// TIA Portal V17 export
// export: Created 2024-06-14T09:53:08.5091314Z, ExportSetting WithDefaults, DisplayName Totally Integrated Automation Portal, DisplayVersion V17, DisplayName TIA Portal Openness, DisplayVersion V17, DisplayName TIA Portal Version Control Interface, DisplayVersion V17, DisplayName Simotion SCOUT TIA, DisplayVersion 5.4.3.0, DisplayName SINAMICS Startdrive Advanced, DisplayVersion V17 SP1 Update 1, DisplayName SINAMICS Startdrive G110M, G120, G120C, G120D, G120P, G115D, DisplayVersion V17 SP1 Update 1, DisplayName SINAMICS Startdrive G130, G150, S120, S150, SINAMICS MV, S210, DisplayVersion V17 SP1 Update 1, DisplayName STEP 7 Professional, DisplayVersion V17, DisplayName STEP 7 Safety, DisplayVersion V17, DisplayName WinCC Professional, DisplayVersion V17
FUNCTION_BLOCK "Check_scale_LPG"   // FB7, LAD
{ S7_Optimized_Access := 'TRUE' }
VERSION : 0.1
// stored: AutoNumber true, IsIECCheckEnabled false, IsRetainMemResEnabled false, MemoryReserve 100, SetENOAutomatically false, UDAEnableTagReadback false
   VAR_INPUT
      Stopper_sesnor : Bool;
      Cylinder_presence : Bool;
      Pass_line_jammer : Bool;
      Down_line_jammer : Bool;
      Start_cycle : Bool;
      Reset_Cycle : Bool;
      Result : Int;
      Pusher : Bool;
      all_fill_done : Bool;
      xResult : Bool;
   END_VAR
   VAR_OUTPUT
      Stopper : Bool;
      LiftTable : Bool;
      Start_Check_Scale : Bool;
      Divider : Bool;
      Reset : Bool;
      CYCLE_ONE : Bool;
   END_VAR
   VAR
      Check_Scale_Started : Bool;
      Lift_Table { S7_SetPoint := 'True'} : TON_TIME;
      PASS : Bool;
      FAIL : Bool;
      LIFT_down { S7_SetPoint := 'True'} : TON_TIME;
      Temp_1 : Int;
      p_trig : Array[0..10] of Bool;
   END_VAR
   VAR RETAIN
      Stopper_count { S7_SetPoint := 'True'} : CTU_INT;
   END_VAR
   VAR
      counter_reset : Bool;
      Scale { S7_SetPoint := 'True'} : TON_TIME;
      Pusher_reset { S7_SetPoint := 'True'} : TON_TIME;
      datasend { ExternalAccessible := 'False'; ExternalVisible := 'False'; ExternalWritable := 'False'} : Bool;
      fb_Fifo_Instance { S7_SetPoint := 'True'} : "fb_Fifo";
      idx7 : Int;
      fb_Compress_Instance { S7_SetPoint := 'True'} : "fb_Compress";
      jammer_on { S7_SetPoint := 'True'} : TON_TIME;
      jammer : Bool;
      pusher_enable : Bool;
      Scale_done : Bool;
   END_VAR
   VAR RETAIN
      Lift_Table_UP { S7_SetPoint := 'True'} : CTU_INT;
   END_VAR
   VAR
      fb_Fifo_Instance_1 { S7_SetPoint := 'True'} : "fb_Fifo";
      fb_Compress_Instance_1 { S7_SetPoint := 'True'} : "fb_Compress";
      timer_1 { S7_SetPoint := 'True'} : TON_TIME;
   END_VAR
   VAR_TEMP
      temp : Int;
   END_VAR
   VAR_TEMP   // added for the SCL form of the ladder/FBD networks
      _w1 : Bool;
      _w2 : Bool;
   END_VAR
BEGIN

REGION Network 1
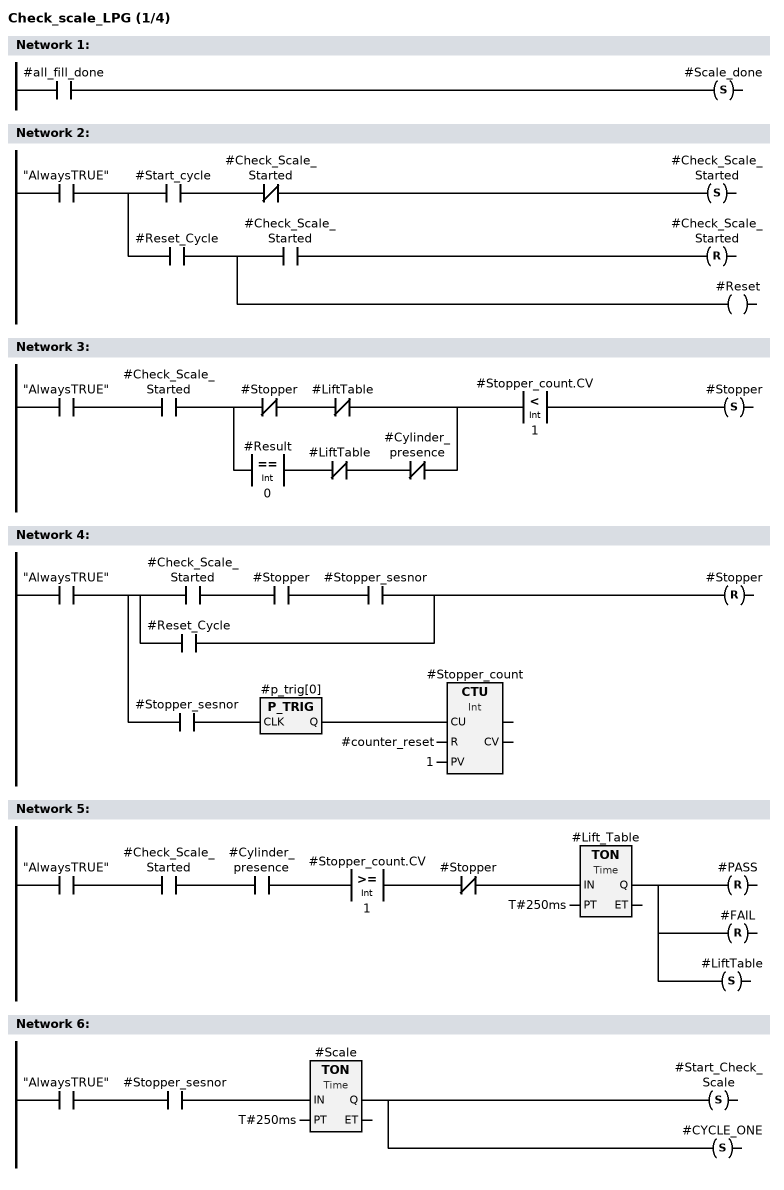
   RUNG wire#powerrail
      Contact( #all_fill_done )
      S_Coil( #Scale_done )
   END_RUNG
   // the same network as SCL:
   IF #all_fill_done THEN #Scale_done := TRUE; END_IF;
END_REGION

REGION Network 2
   RUNG wire#powerrail
      Contact( "AlwaysTRUE" )
      wire#w1
      Contact( #Start_cycle )
      I_Contact( #Check_Scale_Started )
      S_Coil( #Check_Scale_Started )
   END_RUNG
   RUNG wire#w1
      Contact( #Reset_Cycle )
      wire#w2
      Contact( #Check_Scale_Started )
      R_Coil( #Check_Scale_Started )
   END_RUNG
   RUNG wire#w2
      Coil( #Reset )
   END_RUNG
   // the same network as SCL:
   IF "AlwaysTRUE" AND #Start_cycle AND NOT #Check_Scale_Started THEN #Check_Scale_Started := TRUE; END_IF;
   #_w1 := "AlwaysTRUE" AND #Reset_Cycle;
   IF #_w1 AND #Check_Scale_Started THEN #Check_Scale_Started := FALSE; END_IF;
   #Reset := #_w1;
END_REGION

REGION Network 3
   RUNG wire#powerrail
      Contact( "AlwaysTRUE" )
      Contact( #Check_Scale_Started )
      wire#w1
      I_Contact( #Stopper )
      I_Contact( #LiftTable )
      wire#w2
      { S7_Templates := "SrcType := Int" } LT_Contact(in1 := #Stopper_count.CV, in2 := 1)
      S_Coil( #Stopper )
   END_RUNG
   RUNG wire#w1
      { S7_Templates := "SrcType := Int" } EQ_Contact(in1 := #Result, in2 := 0)
      I_Contact( #LiftTable )
      I_Contact( #Cylinder_presence )
   END_RUNG wire#w2
   // the same network as SCL:
   IF "AlwaysTRUE" AND #Check_Scale_Started AND ((NOT #Stopper AND NOT #LiftTable) OR ((#Result = 0) AND NOT #LiftTable AND NOT #Cylinder_presence)) AND (#Stopper_count.CV < 1) THEN
       #Stopper := TRUE;
   END_IF;
END_REGION

REGION Network 4
   RUNG wire#powerrail
      Contact( "AlwaysTRUE" )
      wire#w1
      Contact( #Check_Scale_Started )
      Contact( #Stopper )
      Contact( #Stopper_sesnor )
      wire#w2
      R_Coil( #Stopper )
   END_RUNG
   RUNG wire#w1
      Contact( #Reset_Cycle )
   END_RUNG wire#w2
   RUNG wire#w1
      Contact( #Stopper_sesnor )
      P_Trig( #p_trig[0] )
      { S7_Templates := "value_type := Int" } #Stopper_count.CTU(r := #counter_reset, pv := 1, cv =>)
   END_RUNG
   // the same network as SCL:
   IF "AlwaysTRUE" AND ((#Check_Scale_Started AND #Stopper AND #Stopper_sesnor) OR #Reset_Cycle) THEN
       #Stopper := FALSE;
   END_IF;
   #_w1 := "AlwaysTRUE" AND #Stopper_sesnor;
   #_w2 := #_w1 AND NOT #p_trig[0];   // rising edge
   #p_trig[0] := #_w1;
   #Stopper_count(CU := #_w2, R := #counter_reset, PV := 1);   // CTU
END_REGION

REGION Network 5
   RUNG wire#powerrail
      Contact( "AlwaysTRUE" )
      Contact( #Check_Scale_Started )
      Contact( #Cylinder_presence )
      { S7_Templates := "SrcType := Int" } GE_Contact(in1 := #Stopper_count.CV, in2 := 1)
      I_Contact( #Stopper )
      { S7_Templates := "time_type := Time" } #Lift_Table.TON(pt := T#250ms, et =>)
      wire#w1
      R_Coil( #PASS )
   END_RUNG
   RUNG wire#w1
      R_Coil( #FAIL )
   END_RUNG
   RUNG wire#w1
      S_Coil( #LiftTable )
   END_RUNG
   // the same network as SCL:
   #Lift_Table(IN := "AlwaysTRUE" AND #Check_Scale_Started AND #Cylinder_presence AND (#Stopper_count.CV >= 1) AND NOT #Stopper,   // TON
               PT := T#250ms);
   IF #Lift_Table.Q THEN
       #PASS := FALSE;
       #FAIL := FALSE;
       #LiftTable := TRUE;
   END_IF;
END_REGION

REGION Network 6
   RUNG wire#powerrail
      Contact( "AlwaysTRUE" )
      Contact( #Stopper_sesnor )
      { S7_Templates := "time_type := Time" } #Scale.TON(pt := T#250ms, et =>)
      wire#w1
      S_Coil( #Start_Check_Scale )
   END_RUNG
   RUNG wire#w1
      S_Coil( #CYCLE_ONE )
   END_RUNG
   // the same network as SCL:
   #Scale(IN := "AlwaysTRUE" AND #Stopper_sesnor, PT := T#250ms);   // TON
   IF #Scale.Q THEN
       #Start_Check_Scale := TRUE;
       #CYCLE_ONE := TRUE;
   END_IF;
END_REGION

REGION Network 7
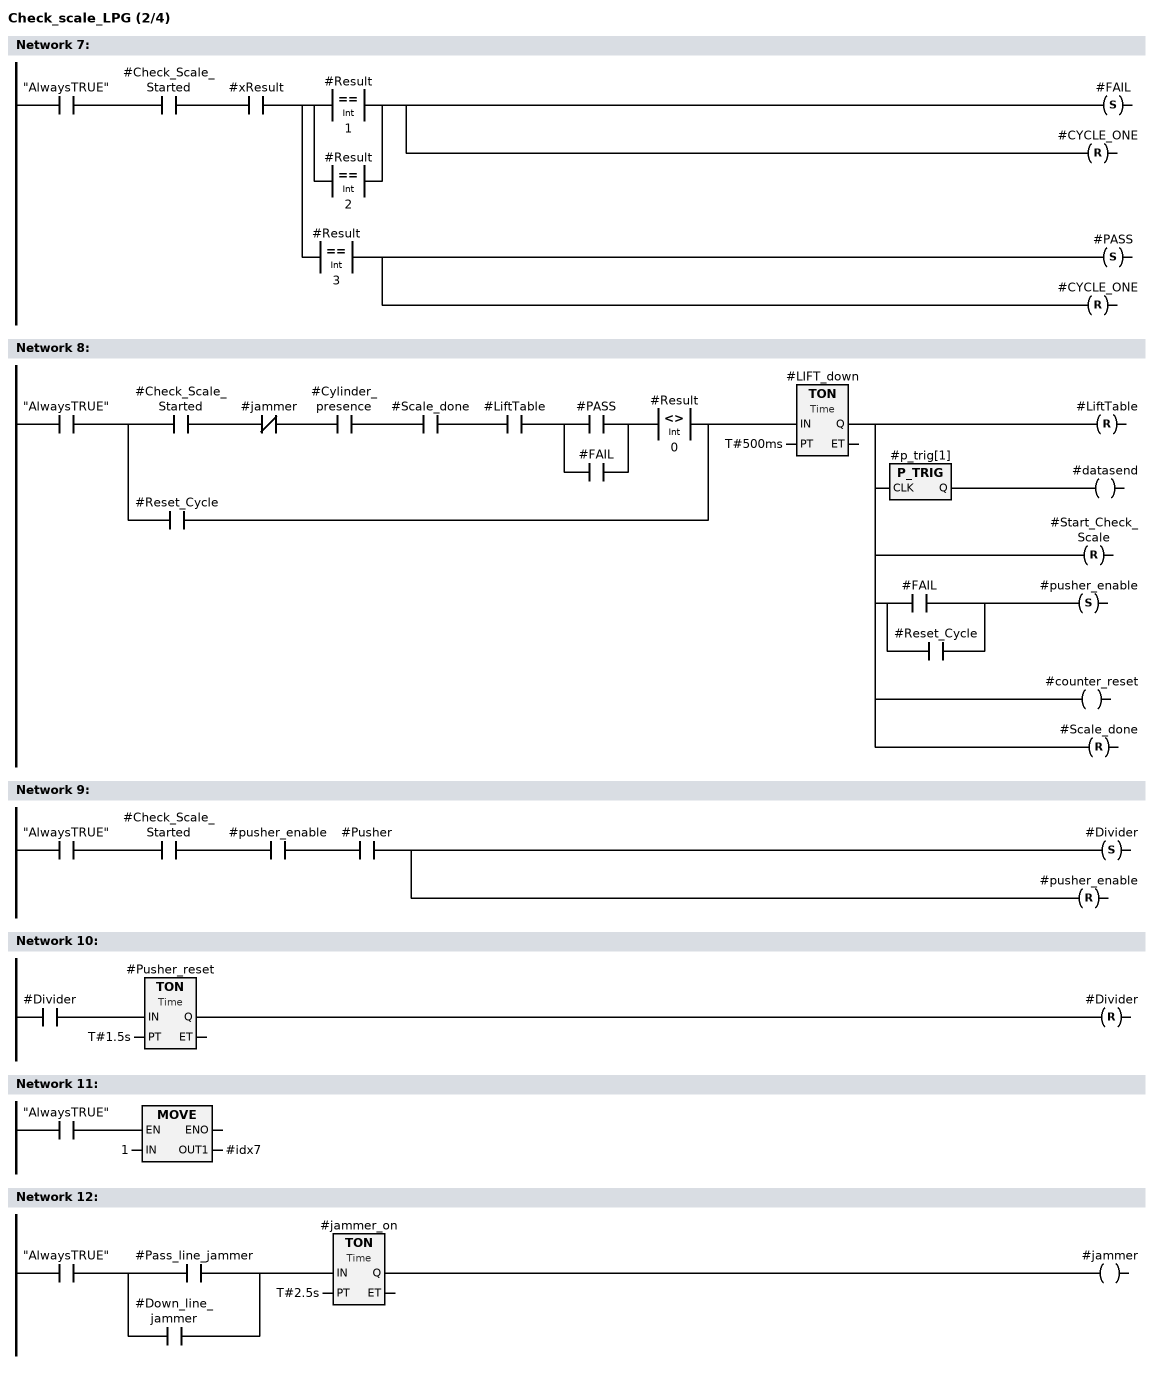
   RUNG wire#powerrail
      Contact( "AlwaysTRUE" )
      Contact( #Check_Scale_Started )
      Contact( #xResult )
      wire#w1
      { S7_Templates := "SrcType := Int" } EQ_Contact(in1 := #Result, in2 := 1)
      wire#w2
      S_Coil( #FAIL )
   END_RUNG
   RUNG wire#w1
      { S7_Templates := "SrcType := Int" } EQ_Contact(in1 := #Result, in2 := 2)
   END_RUNG wire#w2
   RUNG wire#w2
      R_Coil( #CYCLE_ONE )
   END_RUNG
   RUNG wire#w1
      { S7_Templates := "SrcType := Int" } EQ_Contact(in1 := #Result, in2 := 3)
      wire#w3
      S_Coil( #PASS )
   END_RUNG
   RUNG wire#w3
      R_Coil( #CYCLE_ONE )
   END_RUNG
   // the same network as SCL:
   #_w1 := "AlwaysTRUE" AND #Check_Scale_Started AND #xResult;
   IF #_w1 AND ((#Result = 1) OR (#Result = 2)) THEN
       #FAIL := TRUE;
       #CYCLE_ONE := FALSE;
   END_IF;
   IF #_w1 AND (#Result = 3) THEN
       #PASS := TRUE;
       #CYCLE_ONE := FALSE;
   END_IF;
END_REGION

REGION Network 8
   RUNG wire#powerrail
      Contact( "AlwaysTRUE" )
      wire#w1
      Contact( #Check_Scale_Started )
      I_Contact( #jammer )
      Contact( #Cylinder_presence )
      Contact( #Scale_done )
      Contact( #LiftTable )
      wire#w2
      Contact( #PASS )
      wire#w3
      { S7_Templates := "SrcType := Int" } NE_Contact(in1 := #Result, in2 := 0)
      wire#w4
      { S7_Templates := "time_type := Time" } #LIFT_down.TON(pt := T#500ms, et =>)
      wire#w5
      R_Coil( #LiftTable )
   END_RUNG
   RUNG wire#w2
      Contact( #FAIL )
   END_RUNG wire#w3
   RUNG wire#w1
      Contact( #Reset_Cycle )
   END_RUNG wire#w4
   RUNG wire#w5
      P_Trig( #p_trig[1] )
      Coil( #datasend )
   END_RUNG
   RUNG wire#w5
      R_Coil( #Start_Check_Scale )
   END_RUNG
   RUNG wire#w5
      Contact( #FAIL )
      wire#w6
      S_Coil( #pusher_enable )
   END_RUNG
   RUNG wire#w5
      Contact( #Reset_Cycle )
   END_RUNG wire#w6
   RUNG wire#w5
      Coil( #counter_reset )
   END_RUNG
   RUNG wire#w5
      R_Coil( #Scale_done )
   END_RUNG
   // the same network as SCL:
   #LIFT_down(IN := "AlwaysTRUE" AND ((#Check_Scale_Started AND NOT #jammer AND #Cylinder_presence AND #Scale_done AND #LiftTable AND (#PASS OR #FAIL) AND (#Result <> 0)) OR #Reset_Cycle),   // TON
              PT := T#500ms);
   IF #LIFT_down.Q THEN #LiftTable := FALSE; END_IF;
   #_w1 := #LIFT_down.Q AND NOT #p_trig[1];   // rising edge
   #p_trig[1] := #LIFT_down.Q;
   #datasend := #_w1;
   IF #LIFT_down.Q THEN #Start_Check_Scale := FALSE; END_IF;
   IF #LIFT_down.Q AND (#FAIL OR #Reset_Cycle) THEN #pusher_enable := TRUE; END_IF;
   #counter_reset := #LIFT_down.Q;
   IF #LIFT_down.Q THEN #Scale_done := FALSE; END_IF;
END_REGION

REGION Network 9
   RUNG wire#powerrail
      Contact( "AlwaysTRUE" )
      Contact( #Check_Scale_Started )
      Contact( #pusher_enable )
      Contact( #Pusher )
      wire#w1
      S_Coil( #Divider )
   END_RUNG
   RUNG wire#w1
      R_Coil( #pusher_enable )
   END_RUNG
   // the same network as SCL:
   IF "AlwaysTRUE" AND #Check_Scale_Started AND #pusher_enable AND #Pusher THEN
       #Divider := TRUE;
       #pusher_enable := FALSE;
   END_IF;
END_REGION

REGION Network 10
   RUNG wire#powerrail
      Contact( #Divider )
      { S7_Templates := "time_type := Time" } #Pusher_reset.TON(pt := T#1.5s, et =>)
      R_Coil( #Divider )
   END_RUNG
   // the same network as SCL:
   #Pusher_reset(IN := #Divider, PT := T#1.5s);   // TON
   IF #Pusher_reset.Q THEN #Divider := FALSE; END_IF;
END_REGION

REGION Network 11
   RUNG wire#powerrail
      Contact( "AlwaysTRUE" )
      Move(in := 1, out1 => #idx7)
   END_RUNG
   // the same network as SCL:
   IF "AlwaysTRUE" THEN #idx7 := 1; END_IF;
END_REGION

REGION Network 12
   RUNG wire#powerrail
      Contact( "AlwaysTRUE" )
      wire#w1
      Contact( #Pass_line_jammer )
      wire#w2
      { S7_Templates := "time_type := Time" } #jammer_on.TON(pt := T#2.5s, et =>)
      Coil( #jammer )
   END_RUNG
   RUNG wire#w1
      Contact( #Down_line_jammer )
   END_RUNG wire#w2
   // the same network as SCL:
   #jammer_on(IN := "AlwaysTRUE" AND (#Pass_line_jammer OR #Down_line_jammer), PT := T#2.5s);   // TON
   #jammer := #jammer_on.Q;
END_REGION

REGION Network 13: cylinder FAIL
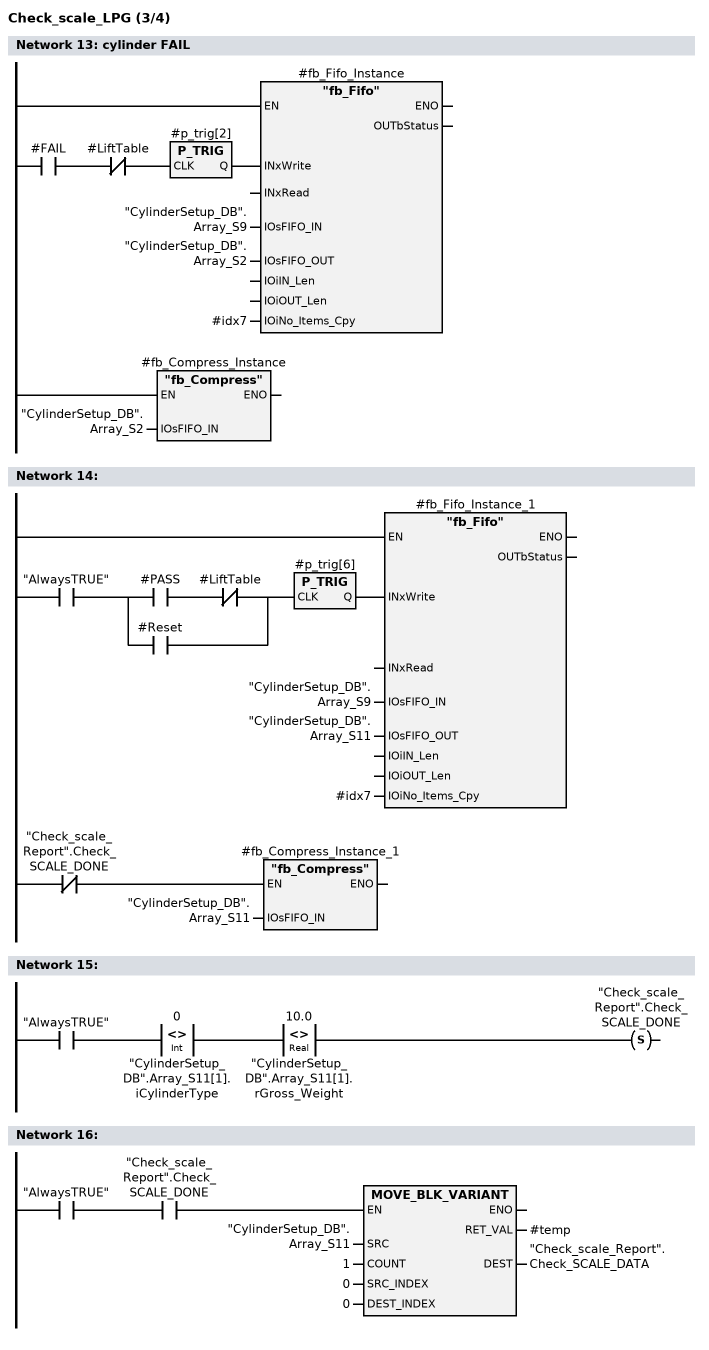
   RUNG wire#powerrail
      #fb_Fifo_Instance(INxWrite := wire#w1, INxRead :=, IOsFIFO_IN := "CylinderSetup_DB".Array_S9, IOsFIFO_OUT := "CylinderSetup_DB".Array_S2, IOiIN_Len :=, IOiOUT_Len :=, IOiNo_Items_Cpy := #idx7, OUTbStatus =>)
   END_RUNG
   RUNG wire#powerrail
      Contact( #FAIL )
      I_Contact( #LiftTable )
      P_Trig( #p_trig[2] )
   END_RUNG wire#w1
   RUNG wire#powerrail
      #fb_Compress_Instance(IOsFIFO_IN := "CylinderSetup_DB".Array_S2)
   END_RUNG
   // the same network as SCL:
   #_w1 := #FAIL AND NOT #LiftTable;
   #_w2 := #_w1 AND NOT #p_trig[2];   // rising edge
   #p_trig[2] := #_w1;
   #fb_Fifo_Instance(INxWrite := #_w2,   // "fb_Fifo"
                     IOsFIFO_IN := "CylinderSetup_DB".Array_S9,
                     IOsFIFO_OUT := "CylinderSetup_DB".Array_S2,
                     IOiNo_Items_Cpy := #idx7);
   #fb_Compress_Instance(IOsFIFO_IN := "CylinderSetup_DB".Array_S2);   // "fb_Compress"
END_REGION

REGION Network 14
   RUNG wire#powerrail
      #fb_Fifo_Instance_1(INxWrite := wire#w3, INxRead :=, IOsFIFO_IN := "CylinderSetup_DB".Array_S9, IOsFIFO_OUT := "CylinderSetup_DB".Array_S11, IOiIN_Len :=, IOiOUT_Len :=, IOiNo_Items_Cpy := #idx7, OUTbStatus =>)
   END_RUNG
   RUNG wire#powerrail
      Contact( "AlwaysTRUE" )
      wire#w1
      Contact( #PASS )
      I_Contact( #LiftTable )
      wire#w2
      P_Trig( #p_trig[6] )
   END_RUNG wire#w3
   RUNG wire#w1
      Contact( #Reset )
   END_RUNG wire#w2
   RUNG wire#powerrail
      I_Contact( "Check_scale_Report".Check_SCALE_DONE )
      #fb_Compress_Instance_1(IOsFIFO_IN := "CylinderSetup_DB".Array_S11)
   END_RUNG
   // the same network as SCL:
   #_w1 := "AlwaysTRUE" AND ((#PASS AND NOT #LiftTable) OR #Reset);
   #_w2 := #_w1 AND NOT #p_trig[6];   // rising edge
   #p_trig[6] := #_w1;
   #fb_Fifo_Instance_1(INxWrite := #_w2,   // "fb_Fifo"
                       IOsFIFO_IN := "CylinderSetup_DB".Array_S9,
                       IOsFIFO_OUT := "CylinderSetup_DB".Array_S11,
                       IOiNo_Items_Cpy := #idx7);
   IF NOT "Check_scale_Report".Check_SCALE_DONE THEN
       #fb_Compress_Instance_1(IOsFIFO_IN := "CylinderSetup_DB".Array_S11);   // "fb_Compress"
   END_IF;
END_REGION

REGION Network 15
   RUNG wire#powerrail
      Contact( "AlwaysTRUE" )
      { S7_Templates := "SrcType := Int" } NE_Contact(in1 := 0, in2 := "CylinderSetup_DB".Array_S11[1].iCylinderType)
      { S7_Templates := "SrcType := Real" } NE_Contact(in1 := 10.0, in2 := "CylinderSetup_DB".Array_S11[1].rGross_Weight)
      S_Coil( "Check_scale_Report".Check_SCALE_DONE )
   END_RUNG
   // the same network as SCL:
   IF "AlwaysTRUE" AND (0 <> "CylinderSetup_DB".Array_S11[1].iCylinderType) AND (10.0 <> "CylinderSetup_DB".Array_S11[1].rGross_Weight) THEN
       "Check_scale_Report".Check_SCALE_DONE := TRUE;
   END_IF;
END_REGION

REGION Network 16
   RUNG wire#powerrail
      Contact( "AlwaysTRUE" )
      Contact( "Check_scale_Report".Check_SCALE_DONE )
      MOVE_BLK_VARIANT(SRC := "CylinderSetup_DB".Array_S11, COUNT := 1, SRC_INDEX := 0, DEST_INDEX := 0, Ret_Val => #temp, DEST => "Check_scale_Report".Check_SCALE_DATA)
   END_RUNG
   // the same network as SCL:
   IF "AlwaysTRUE" AND "Check_scale_Report".Check_SCALE_DONE THEN
       #temp := MOVE_BLK_VARIANT(SRC := "CylinderSetup_DB".Array_S11,
                               COUNT := 1,
                               SRC_INDEX := 0,
                               DEST_INDEX := 0,
                               DEST => "Check_scale_Report".Check_SCALE_DATA);
   END_IF;
END_REGION

REGION Network 17
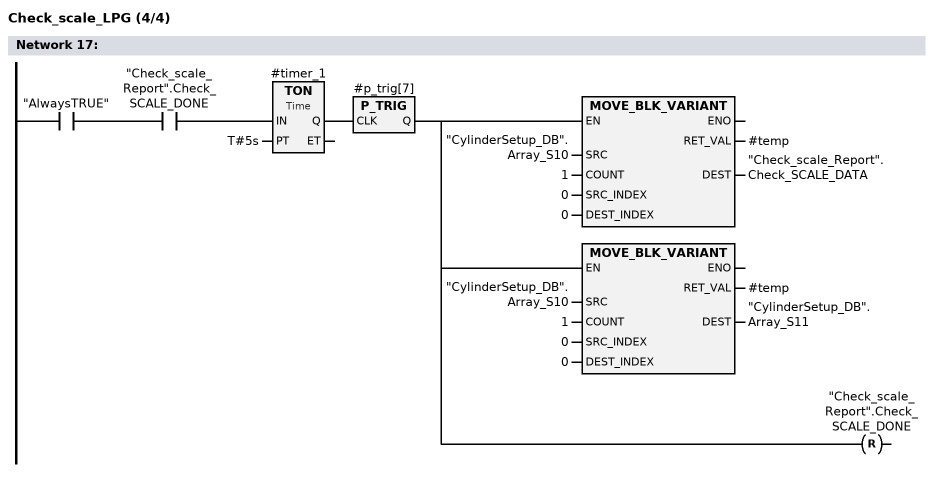
   RUNG wire#powerrail
      Contact( "AlwaysTRUE" )
      Contact( "Check_scale_Report".Check_SCALE_DONE )
      { S7_Templates := "time_type := Time" } #timer_1.TON(pt := T#5s, et =>)
      P_Trig( #p_trig[7] )
      wire#w1
      MOVE_BLK_VARIANT(SRC := "CylinderSetup_DB".Array_S10, COUNT := 1, SRC_INDEX := 0, DEST_INDEX := 0, Ret_Val => #temp, DEST => "Check_scale_Report".Check_SCALE_DATA)
   END_RUNG
   RUNG wire#w1
      MOVE_BLK_VARIANT(SRC := "CylinderSetup_DB".Array_S10, COUNT := 1, SRC_INDEX := 0, DEST_INDEX := 0, Ret_Val => #temp, DEST => "CylinderSetup_DB".Array_S11)
   END_RUNG
   RUNG wire#w1
      R_Coil( "Check_scale_Report".Check_SCALE_DONE )
   END_RUNG
   // the same network as SCL:
   #timer_1(IN := "AlwaysTRUE" AND "Check_scale_Report".Check_SCALE_DONE, PT := T#5s);   // TON
   #_w1 := #timer_1.Q AND NOT #p_trig[7];   // rising edge
   #p_trig[7] := #timer_1.Q;
   IF #_w1 THEN
       #temp := MOVE_BLK_VARIANT(SRC := "CylinderSetup_DB".Array_S10,
                               COUNT := 1,
                               SRC_INDEX := 0,
                               DEST_INDEX := 0,
                               DEST => "Check_scale_Report".Check_SCALE_DATA);
       #temp := MOVE_BLK_VARIANT(SRC := "CylinderSetup_DB".Array_S10,
                               COUNT := 1,
                               SRC_INDEX := 0,
                               DEST_INDEX := 0,
                               DEST => "CylinderSetup_DB".Array_S11);
       "Check_scale_Report".Check_SCALE_DONE := FALSE;
   END_IF;
END_REGION
END_FUNCTION_BLOCK
